// TIA Portal V20 export
// export: Created 2026-08-26T00:00:00.0000000Z, ExportSetting WithDefaults, DisplayName Totally Integrated Automation Portal, DisplayVersion V20, DisplayName TIA Portal Openness, DisplayVersion V20, DisplayName STEP 7 Professional, DisplayVersion V20
DATA_BLOCK "Diag_DB"   // DB
{ S7_Optimized_Access := 'TRUE' }
VERSION : 0.1
// Station health, written by OB86 (RackOrStationFailure). Until this existed, an ET200SP could lose power and nothing in the system noticed: the valves on it simply stopped answering while the HMI carried on showing their last known positions as though they were live. Stale data presented as current is the actual hazard here, more than the loss of control - an operator plans a ballast transfer on positions that stopped being true ten minutes ago. The three hardware identifiers are data rather than code so that re-adding a station in TIA, which reassigns them, does not require an SCL edit. Read the current values off the SYSTEM DIAGNOSTICS screen: every device tile shows its identifier beneath the name.
// stored: AutoNumber true, IsOnlyStoredInLoadMemory false, IsRetainMemResEnabled false, IsWriteProtectedInAS false, MemoryReserve 100
   VAR
      Laddr_AFT : UInt := 273;   // Hardware identifier of ET200SP_AFT. Read off the SYSTEM DIAGNOSTICS screen - each device tile shows it under the name. Held here rather than in OB86 so that re-adding a station in TIA, which reassigns identifiers, is a data change and not a code change.
      Laddr_MID : UInt := 288;   // Hardware identifier of ET200SP_MID.
      Laddr_FWD : UInt := 306;   // Hardware identifier of ET200SP_FWD.
      AftLost : Bool;   // ET200SP_AFT is off the network. Valves 1-27 are unreachable and whatever the HMI shows for them is stale.
      MidLost : Bool;   // ET200SP_MID is off the network. Valves 28-54 are unreachable.
      FwdLost : Bool;   // ET200SP_FWD is off the network. Valves 55-89 are unreachable.
      UnknownLost : Bool;   // A station failed whose hardware identifier matches none of the three above. Means either the identifiers were reassigned and this DB was not updated, or a device exists that OB86 does not know about. Never silently ignored - that would hide a real station failure.
      AnyStationLost : Bool;   // Any of the four flags above. One bit for a screen to watch instead of ORing four.
      LastUnknownLaddr : UInt;   // The unrecognised identifier, kept so it can be looked up on the SYSTEM DIAGNOSTICS screen rather than guessed at.
      AftLossCount : Int;   // How many times AFT has dropped since startup. A station that is cleanly down reads 1; one that is flapping on a bad cable or a loose connector climbs, and that difference does not show in the status bit alone.
      MidLossCount : Int;   // Drop count for MID.
      FwdLossCount : Int;   // Drop count for FWD.
      ModuleFault : Bool;   // LATCHED: an I/O module raised a diagnostic. Cleared only by ModuleFaultAck - never self-clearing, see OB82.
      ModuleFaultAck : Bool;   // Write TRUE to clear ModuleFault. FB_ValveLoop consumes and clears this.
      ModuleEventCount : Int;   // Total OB82 events since CPU start. Rising with no new fault = a module chattering.
      LastModuleLaddr : UInt;   // Hardware identifier from the most recent OB82 event - identifies WHICH module.
      LastModuleIoState : Word;   // Raw IO_State word from the most recent OB82 event. Stored undecoded on purpose.
      LastModuleChannel : UInt;   // Channel number from the most recent OB82 event - narrows a fault to one terminal.
      LastModuleMultiError : Bool;   // TRUE if that event carried more than one error.
      NewModuleEvent : Bool;   // Set by OB82, consumed by FB_ValveLoop. The decode deliberately lives in FB_ValveLoop, not OB82, so it can be tested from a watch table - OB82 itself cannot be triggered in PLCSIM.
      ModuleLaddr : Array[1..36] of UInt;   // Hardware identifier of each I/O module, read from the PLC system constants 2026-09-10. Index order is RACK order: 1-11 AFT slots 1-11, 12-22 MID slots 1-11, 23-36 FWD slots 1-14. Held as DATA, not literals in SCL, for the same reason as Laddr_AFT/MID/FWD above. WARNING: re-adding a module in TIA reassigns these, and a shifted table would name the WRONG module - the unknown handler only catches a MISSING entry. Re-read the system constants after any hardware change. Note AFT is not contiguous (DQ ST_1 is 281, between the DI values) so a range check cannot substitute for this table.
      W_ModuleFault : Array[0..2] of Word;   // One LATCHED bit per I/O module. Module index i (1..36) is word (i-1)/16, bit (i-1) MOD 16 - the same packing the valve alarm words use. Cleared only by ModuleFaultAck.
      UnknownModuleFault : Bool;   // An OB82 event arrived whose LADDR is not in ModuleLaddr[]. Means the table is stale or an unexpected device reported. Never silently dropped.
      UnknownModuleLaddr : UInt;   // The unrecognised identifier, so a stale table can be diagnosed.
   END_VAR
BEGIN
   ModuleLaddr[1] := 280;
   ModuleLaddr[2] := 282;
   ModuleLaddr[3] := 283;
   ModuleLaddr[4] := 284;
   ModuleLaddr[5] := 285;
   ModuleLaddr[6] := 286;
   ModuleLaddr[7] := 287;
   ModuleLaddr[8] := 281;
   ModuleLaddr[9] := 270;
   ModuleLaddr[10] := 271;
   ModuleLaddr[11] := 272;
   ModuleLaddr[12] := 295;
   ModuleLaddr[13] := 296;
   ModuleLaddr[14] := 297;
   ModuleLaddr[15] := 298;
   ModuleLaddr[16] := 299;
   ModuleLaddr[17] := 300;
   ModuleLaddr[18] := 301;
   ModuleLaddr[19] := 302;
   ModuleLaddr[20] := 303;
   ModuleLaddr[21] := 304;
   ModuleLaddr[22] := 305;
   ModuleLaddr[23] := 313;
   ModuleLaddr[24] := 314;
   ModuleLaddr[25] := 315;
   ModuleLaddr[26] := 316;
   ModuleLaddr[27] := 317;
   ModuleLaddr[28] := 318;
   ModuleLaddr[29] := 319;
   ModuleLaddr[30] := 320;
   ModuleLaddr[31] := 321;
   ModuleLaddr[32] := 322;
   ModuleLaddr[33] := 323;
   ModuleLaddr[34] := 324;
   ModuleLaddr[35] := 325;
   ModuleLaddr[36] := 326;
END_DATA_BLOCK
